FUNCTION_BLOCK Mover IMPLEMENTS I_Mover
VAR CONSTANT
	MAX_DATA : INT := 10;
END_VAR
VAR
	_axisRef 	: AXIS_REF;
	//_linkID		: UDINT;
	_IPos		: I_PosMover;
	_position	: LREAL;
	_IMode		: I_Mode;
	_ID			: UDINT;
	_step		: UDINT;
	_data		: ARRAY [1..MAX_DATA] OF LREAL;
	_target		: LREAL;
END_VAR

METHOD ChangeStep : BOOL
VAR_INPUT
	step	: UDINT;
END_VAR
_step := step;
END_METHOD

METHOD Cyclic : BOOL
VAR
	inTargetPos : BOOL;
	tolerance : LREAL := 1.0;
END_VAR
// In Target Position
inTargetPos := FALSE;
IF (ABS(_target - position) < tolerance) THEN
	inTargetPos := TRUE;
END_IF
 
// Move
IF _IMode.Mode = E_Mode.automatic AND NOT inTargetPos THEN
	_position := _position + 0.6;
	IF _position > 3000 THEN
		_position := _position - 3000;
	END_IF
END_IF

IF _Ipos <> 0 THEN
	_target := _IPos.TargetPosition;	
END_IF
END_METHOD

{warning 'Add property implementation'}
PROPERTY ErrorCode : UDINT
GET
END_GET
END_PROPERTY

//FB_Init is always available implicitly and it is used primarily for initialization.
//The return value is not evaluated. For a specific influence, you can also declare the
//methods explicitly and provide additional code there with the standard initialization
//code. You can evaluate the return value.
METHOD FB_Init: BOOL
VAR_INPUT
    bInitRetains: BOOL; // TRUE: the retain variables are initialized (reset warm / reset cold)
    bInCopyCode: BOOL;  // TRUE: the instance will be copied to the copy code afterward (online change)
	ID : UDINT;   
	mode : I_Mode;
	manager : I_RegisterMover;
END_VAR
manager.RegisterMover(THIS^);
_ID := ID;
_IMode := mode;
END_METHOD

{warning 'Add property implementation'}
PROPERTY ID : UDINT
GET
ID := _ID;
END_GET
END_PROPERTY

{warning 'Add property implementation'}
PROPERTY Linked : BOOL
GET
Linked := _IPos <> 0;
END_GET
END_PROPERTY

METHOD MoveToPosition : BOOL
VAR_INPUT
END_VAR
END_METHOD

{warning 'Add property implementation'}
PROPERTY Position : LREAL
GET
Position := _position;
END_GET
SET
END_SET
END_PROPERTY

METHOD SetData : BOOL
VAR_INPUT
	index	: INT;
	value	: LREAL;
END_VAR
IF index > 0 AND index <= MAX_DATA THEN
	_data[index] := value;
END_IF
END_METHOD

METHOD SetPosLink : BOOL
VAR_INPUT
	position : I_PosMover;
END_VAR
_IPos := position;
END_METHOD

{warning 'Add property implementation'}
PROPERTY State : UDINT
GET
END_GET
SET
END_SET
END_PROPERTY

{warning 'Add property implementation'}
PROPERTY Step : UDINT
GET
Step := _step;
END_GET
END_PROPERTY

{warning 'Add method implementation '}
METHOD Unlink : BOOL
END_METHOD

{warning 'Add method implementation '}
METHOD Update : BOOL
END_METHOD

END_FUNCTION_BLOCK

(* stored: Version 1.1.0.1
   POU Mover: Id {2359cc95-eb1f-475f-950f-0dd4a4dc4b14}, SpecialFunc None
   Method ChangeStep: Id {6c31488f-ae21-4f22-bdbe-fbb9896ed374}
   Method Cyclic: Id {af42b007-9481-4d60-8aea-f12e455d43b4}
   Property ErrorCode: Id {43598883-c1ad-4d69-88bd-386a6508db73}
   Get Get: Id {442ae90c-0a1e-4fe6-9410-98474ad5adca}
   Method FB_Init: Id {e070e80c-a14f-42d7-b5ae-7b92c470e50f}
   Property ID: Id {46a55ecd-0158-4dcf-bea7-8f329bd5171d}
   Get Get: Id {d4dee1fa-cbc0-4ce7-814c-98b4e4b91309}
   Property Linked: Id {f3c2b9b4-f6e9-4eeb-8509-e8f3267d44ec}
   Get Get: Id {7e8d3845-7dde-4499-90dc-d0456b2f12eb}
   Method MoveToPosition: Id {9e38c854-2c62-4431-9b32-6c8a8ab5d1e2}
   Property Position: Id {4747cc7e-25fa-4479-812a-079d3dcef86c}
   Get Get: Id {d36d252f-9908-4ada-b130-442016ad99ec}
   Set Set: Id {fd34e7f1-c4c8-4c56-9aa9-fac754e7f2f4}
   Method SetData: Id {6b05eac9-b6ae-403d-b1ac-0557c6c55cc9}
   Method SetPosLink: Id {e326a7de-0da8-46b3-8aed-32b5881f8054}
   Property State: Id {ed9ce5fd-b36d-443b-9f70-ad967b07e4d3}
   Get Get: Id {aca6adcf-44da-49f7-8589-e646b8c20af0}
   Set Set: Id {f7040f92-e8a7-4cf9-a6ce-b80286f04bff}
   Property Step: Id {10920e3b-a3f2-41f7-8aeb-fa638111eb52}
   Get Get: Id {42f9d3e3-efe2-46b0-9f7d-b1dbef6e632b}
   Method Unlink: Id {9551b306-a16c-4828-8465-3eb59dac4683}
   Method Update: Id {a9dc30dd-bfe3-4f0a-94fc-779ede3e86c8} *)
